PROGRAM POU_DT02_MotorControl
VAR
	
	fbHaltLeftMotor			: MC_Halt;
	fbHaltRightMotor		: MC_Halt;
	fbJogLeftMotor			: MC_Jog;
	fbJogRightMotor			: MC_Jog;
	testOnlineEdit			: BOOL;
	
END_VAR

IF NOT SystemON THEN
	
	HaltLeftMotor 			:= TRUE;
	HaltRightMotor 			:= TRUE;
	JogLeftMotor 			:= FALSE;
	JogRightMotor 			:= FALSE;
	
ELSE
	
	IF LeftLimitExceeded THEN
		
		HaltLeftMotor 		:= TRUE;
		JogLeftMotor 		:= FALSE;
		
	ELSE
		
		HaltLeftMotor 		:= FALSE;
		JogLeftMotor 		:= TRUE;
		
	END_IF
		
	IF RightLimitExceeded THEN
		
		HaltRightMotor 		:= TRUE;
		JogRightMotor 		:= FALSE;
		
	ELSE
		
		HaltRightMotor 		:= FALSE;
		JogRightMotor 		:= TRUE;
		
	END_IF
IF TRUE THEN
    testOnlineEdit			:= TRUE;
END_IF
	
END_IF

fbHaltLeftMotor(
	Axis					:= LeftMotor,
	Execute					:= HaltLeftMotor);
	
fbHaltRightMotor(
	Axis					:= RightMotor,
	Execute					:= HaltRightMotor);

fbJogLeftMotor(
	Axis					:= LeftMotor,
	JogForward				:= JogLeftMotor,
	Velocity				:= 500.0,
	Acceleration			:= 250.0,
	Deceleration			:= 500.0,
	Mode					:= E_JogMode.MC_JOGMODE_CONTINOUS);
	
fbJogRightMotor(
	Axis					:= RightMotor,
	JogForward				:= JogRightMotor,
	Velocity				:= 500.0,
	Acceleration			:= 250.0,
	Deceleration			:= 500.0,
	Mode					:= E_JogMode.MC_JOGMODE_CONTINOUS);

END_PROGRAM

(* stored: Version 1.1.0.1, ProductVersion 3.1.4022.7
   POU POU_DT02_MotorControl: Id {4c9b7adf-695a-4329-8669-b200073d6e6c}, SpecialFunc None *)
